% RSLogix 500 project PROJECT10- PUMP PROTECTION.RSS, saved by version 8.30.00.16 %
PROJECT "UNTITLED"    % processor: Bul.1763 MicroLogix 1100 Series B %

PROGRAM FILES
  LAD 2 "MAIN"  5 rungs
  LAD 3 "IO"  8 rungs
  LAD 4 "ALARMS"  9 rungs
  LAD 5 "CTRL"  7 rungs
  LAD 6 "HOA"  6 rungs

DATA FILES
  O0 OUTPUT  4 elements
  I1 INPUT  6 elements
  S2 STATUS  66 elements
  B3 BINARY  2 elements
  T4 TIMER  4 elements
  C5 COUNTER  1 elements
  R6 CONTROL  1 elements
  N7 INTEGER  3 elements
  F8 FLOAT  1 elements

LADDER 2 "MAIN"
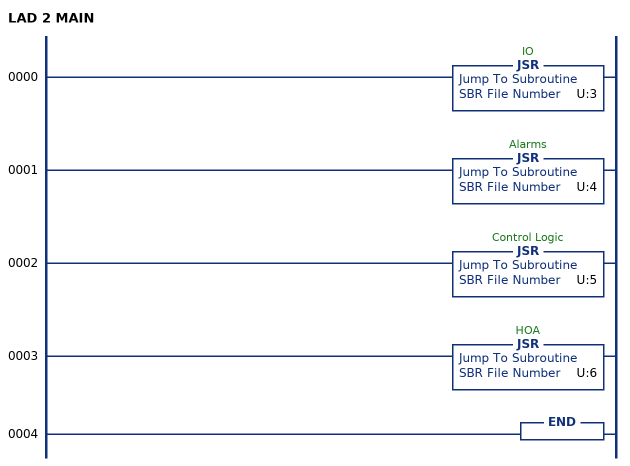
% Rung: 0 %
SOR JSR U:3 EOR
%   U:3  "IO" %
% Rung: 1 %
SOR JSR U:4 EOR
%   U:4  "Alarms" %
% Rung: 2 %
SOR JSR U:5 EOR
%   U:5  "Control Logic" %
% Rung: 3 %
SOR JSR U:6 EOR
%   U:6  "HOA" %
% Rung: 4 %
SOR END EOR

LADDER 3 "IO"
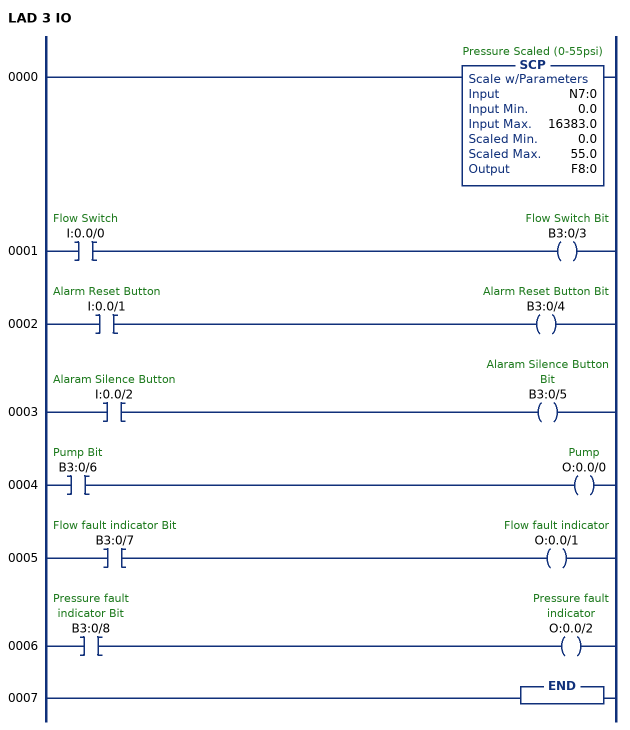
% Rung: 0 %
SOR SCP N7:0 0.0 16383.0 0.0 55.0 F8:0 EOR
%   N7:0  "Pressure Sensor Input" %
%   F8:0  "Pressure Scaled (0-55psi)" %
% Rung: 1 %
SOR XIC I:0.0/0 OTE B3:0/3 EOR
%   I:0.0/0  "Flow Switch" %
%   B3:0/3  "Flow Switch Bit" %
% Rung: 2 %
SOR XIC I:0.0/1 OTE B3:0/4 EOR
%   I:0.0/1  "Alarm Reset Button" %
%   B3:0/4  "Alarm Reset Button Bit" %
% Rung: 3 %
SOR XIC I:0.0/2 OTE B3:0/5 EOR
%   I:0.0/2  "Alaram Silence Button" %
%   B3:0/5  "Alaram Silence Button Bit" %
% Rung: 4 %
SOR XIC B3:0/6 OTE O:0.0/0 EOR
%   B3:0/6  "Pump Bit" %
%   O:0.0/0  "Pump" %
% Rung: 5 %
SOR XIC B3:0/7 OTE O:0.0/1 EOR
%   B3:0/7  "Flow fault indicator Bit" %
%   O:0.0/1  "Flow fault indicator" %
% Rung: 6 %
SOR XIC B3:0/8 OTE O:0.0/2 EOR
%   B3:0/8  "Pressure fault indicator Bit" %
%   O:0.0/2  "Pressure fault indicator" %
% Rung: 7 %
SOR END EOR

LADDER 4 "ALARMS"
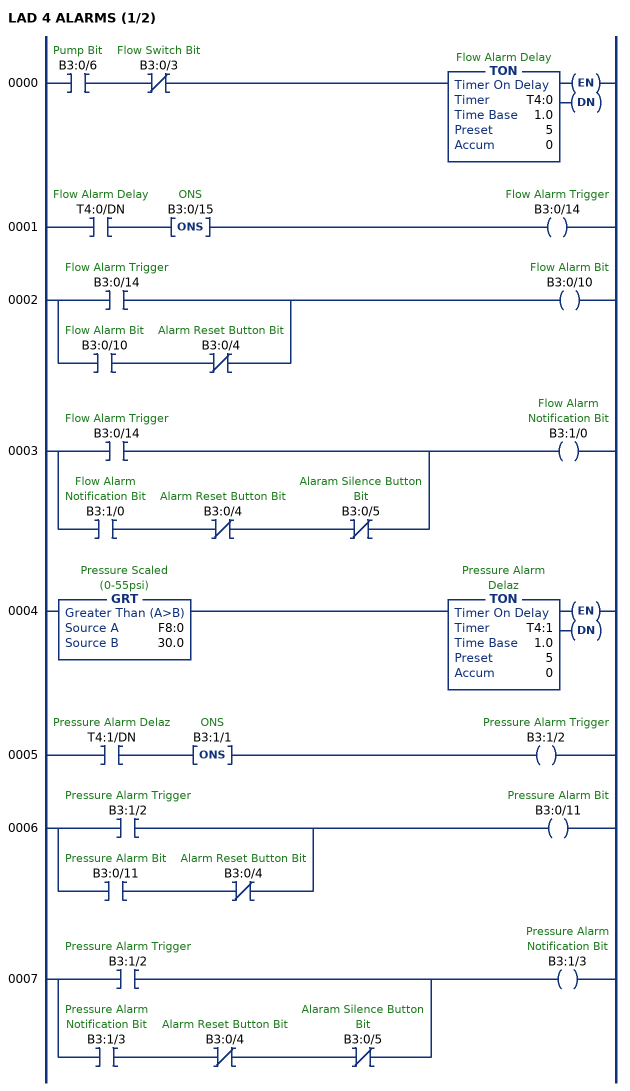
% Rung: 0 %
SOR XIC B3:0/6 XIO B3:0/3 TON T4:0 1.0 5 0 EOR
%   B3:0/6  "Pump Bit" %
%   B3:0/3  "Flow Switch Bit" %
%   T4:0  "Flow Alarm Delay" %
% Rung: 1 %
SOR XIC T4:0/DN ONS B3:0/15 OTE B3:0/14 EOR
%   T4:0  "Flow Alarm Delay" %
%   B3:0/15  "ONS" %
%   B3:0/14  "Flow Alarm Trigger" %
% Rung: 2 %
SOR BST XIC B3:0/14 NXB XIC B3:0/10 XIO B3:0/4 BND OTE B3:0/10 EOR
%   B3:0/14  "Flow Alarm Trigger" %
%   B3:0/10  "Flow Alarm Bit" %
%   B3:0/4  "Alarm Reset Button Bit" %
% Rung: 3 %
SOR BST XIC B3:0/14 NXB XIC B3:1/0 XIO B3:0/4 XIO B3:0/5 BND OTE B3:1/0 EOR
%   B3:0/14  "Flow Alarm Trigger" %
%   B3:1/0  "Flow Alarm Notification Bit" %
%   B3:0/4  "Alarm Reset Button Bit" %
%   B3:0/5  "Alaram Silence Button Bit" %
% Rung: 4 %
SOR GRT F8:0 30.0 TON T4:1 1.0 5 0 EOR
%   F8:0  "Pressure Scaled (0-55psi)" %
%   T4:1  "Pressure Alarm Delaz" %
% Rung: 5 %
SOR XIC T4:1/DN ONS B3:1/1 OTE B3:1/2 EOR
%   T4:1  "Pressure Alarm Delaz" %
%   B3:1/1  "ONS" %
%   B3:1/2  "Pressure Alarm Trigger" %
% Rung: 6 %
SOR BST XIC B3:1/2 NXB XIC B3:0/11 XIO B3:0/4 BND OTE B3:0/11 EOR
%   B3:1/2  "Pressure Alarm Trigger" %
%   B3:0/11  "Pressure Alarm Bit" %
%   B3:0/4  "Alarm Reset Button Bit" %
% Rung: 7 %
SOR BST XIC B3:1/2 NXB XIC B3:1/3 XIO B3:0/4 XIO B3:0/5 BND OTE B3:1/3 EOR
%   B3:1/2  "Pressure Alarm Trigger" %
%   B3:1/3  "Pressure Alarm Notification Bit" %
%   B3:0/4  "Alarm Reset Button Bit" %
%   B3:0/5  "Alaram Silence Button Bit" %

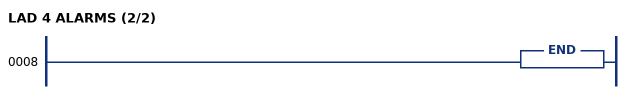
% Rung: 8 %
SOR END EOR

LADDER 5 "CTRL"
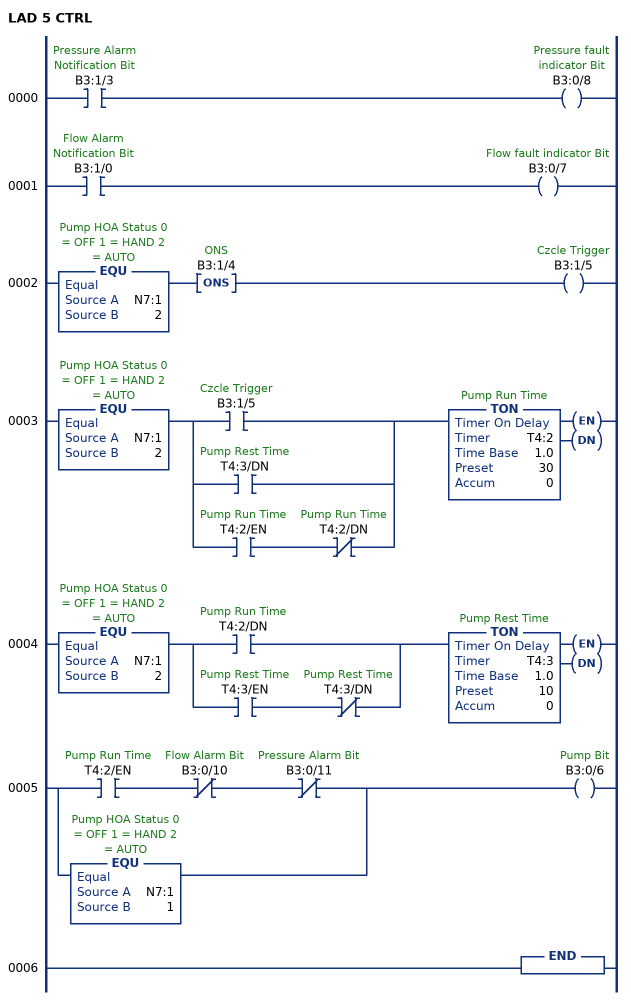
% Rung: 0 %
SOR XIC B3:1/3 OTE B3:0/8 EOR
%   B3:1/3  "Pressure Alarm Notification Bit" %
%   B3:0/8  "Pressure fault indicator Bit" %
% Rung: 1 %
SOR XIC B3:1/0 OTE B3:0/7 EOR
%   B3:1/0  "Flow Alarm Notification Bit" %
%   B3:0/7  "Flow fault indicator Bit" %
% Rung: 2 %
SOR EQU N7:1 2 ONS B3:1/4 OTE B3:1/5 EOR
%   N7:1  "Pump HOA Status 0 = OFF 1 = HAND 2 = AUTO" %
%   B3:1/4  "ONS" %
%   B3:1/5  "Czcle Trigger" %
% Rung: 3 %
SOR EQU N7:1 2 BST BST XIC B3:1/5 NXB XIC T4:3/DN BND NXB XIC T4:2/EN XIO T4:2/DN BND TON T4:2 1.0 30 0 EOR
%   N7:1  "Pump HOA Status 0 = OFF 1 = HAND 2 = AUTO" %
%   B3:1/5  "Czcle Trigger" %
%   T4:3  "Pump Rest Time" %
%   T4:2  "Pump Run Time" %
% Rung: 4 %
SOR EQU N7:1 2 BST XIC T4:2/DN NXB XIC T4:3/EN XIO T4:3/DN BND TON T4:3 1.0 10 0 EOR
%   N7:1  "Pump HOA Status 0 = OFF 1 = HAND 2 = AUTO" %
%   T4:2  "Pump Run Time" %
%   T4:3  "Pump Rest Time" %
% Rung: 5 %
SOR BST XIC T4:2/EN XIO B3:0/10 XIO B3:0/11 NXB EQU N7:1 1 BND OTE B3:0/6 EOR
%   T4:2  "Pump Run Time" %
%   B3:0/10  "Flow Alarm Bit" %
%   B3:0/11  "Pressure Alarm Bit" %
%   N7:1  "Pump HOA Status 0 = OFF 1 = HAND 2 = AUTO" %
%   B3:0/6  "Pump Bit" %
% Rung: 6 %
SOR END EOR

LADDER 6 "HOA"
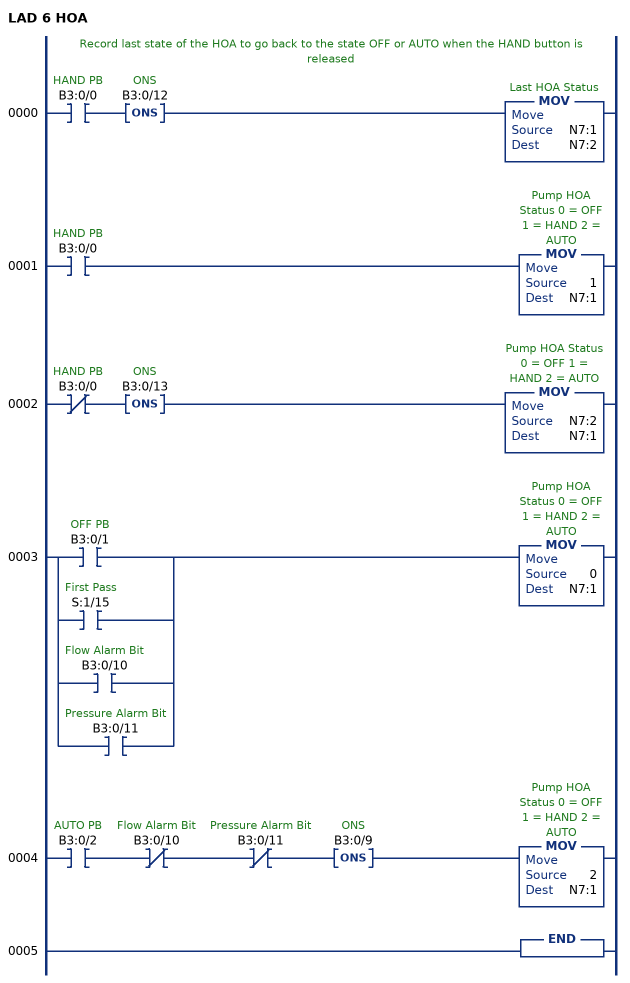
% Rung: 0 %
% Record last state of the HOA to go back to the state OFF or AUTO when the HAND button is released %
SOR XIC B3:0/0 ONS B3:0/12 MOV N7:1 N7:2 EOR
%   B3:0/0  "HAND PB" %
%   B3:0/12  "ONS" %
%   N7:1  "Pump HOA Status 0 = OFF 1 = HAND 2 = AUTO" %
%   N7:2  "Last HOA Status" %
% Rung: 1 %
SOR XIC B3:0/0 MOV 1 N7:1 EOR
%   B3:0/0  "HAND PB" %
%   N7:1  "Pump HOA Status 0 = OFF 1 = HAND 2 = AUTO" %
% Rung: 2 %
SOR XIO B3:0/0 ONS B3:0/13 MOV N7:2 N7:1 EOR
%   B3:0/0  "HAND PB" %
%   B3:0/13  "ONS" %
%   N7:2  "Last HOA Status" %
%   N7:1  "Pump HOA Status 0 = OFF 1 = HAND 2 = AUTO" %
% Rung: 3 %
SOR BST XIC B3:0/1 NXB XIC S:1/15 NXB XIC B3:0/10 NXB XIC B3:0/11 BND MOV 0 N7:1 EOR
%   B3:0/1  "OFF PB" %
%   S:1/15  "First Pass" %
%   B3:0/10  "Flow Alarm Bit" %
%   B3:0/11  "Pressure Alarm Bit" %
%   N7:1  "Pump HOA Status 0 = OFF 1 = HAND 2 = AUTO" %
% Rung: 4 %
SOR XIC B3:0/2 XIO B3:0/10 XIO B3:0/11 ONS B3:0/9 MOV 2 N7:1 EOR
%   B3:0/2  "AUTO PB" %
%   B3:0/10  "Flow Alarm Bit" %
%   B3:0/11  "Pressure Alarm Bit" %
%   B3:0/9  "ONS" %
%   N7:1  "Pump HOA Status 0 = OFF 1 = HAND 2 = AUTO" %
% Rung: 5 %
SOR END EOR

DATA TABLE (non-zero values as saved)
DATA B3
% B3:0 % 0X2048 0X0010
DATA T4
% .PRE .ACC %
% T4:0 % 5 0
% T4:1 % 5 0
% T4:2 % 30 0
% T4:3 % 10 0
DATA N7
% N7:0 % 8192 2 0
DATA F8
% F8:0 % 27.50168
